// SIMATIC STEP 7 (V5.x) project Bai2_PLC

ORGANIZATION_BLOCK OB 1
TITLE = "Main Program Sweep (Cycle)"
VERSION : 0.1
VAR_TEMP
  OB1_EV_CLASS : BYTE ;	//Bits 0-3 = 1 (Coming event), Bits 4-7 = 1 (Event class 1)
  OB1_SCAN_1 : BYTE ;	//1 (Cold restart scan 1 of OB 1), 3 (Scan 2-n of OB 1)
  OB1_PRIORITY : BYTE ;	//Priority of OB Execution
  OB1_OB_NUMBR : BYTE ;	//1 (Organization block 1, OB1)
  OB1_RESERVED_1 : BYTE ;	//Reserved for system
  OB1_RESERVED_2 : BYTE ;	//Reserved for system
  OB1_PREV_CYCLE : INT ;	//Cycle time of previous OB1 scan (milliseconds)
  OB1_MIN_CYCLE : INT ;	//Minimum cycle time of OB1 (milliseconds)
  OB1_MAX_CYCLE : INT ;	//Maximum cycle time of OB1 (milliseconds)
  OB1_DATE_TIME : DATE_AND_TIME ;	//Date and time OB1 started
END_VAR
BEGIN
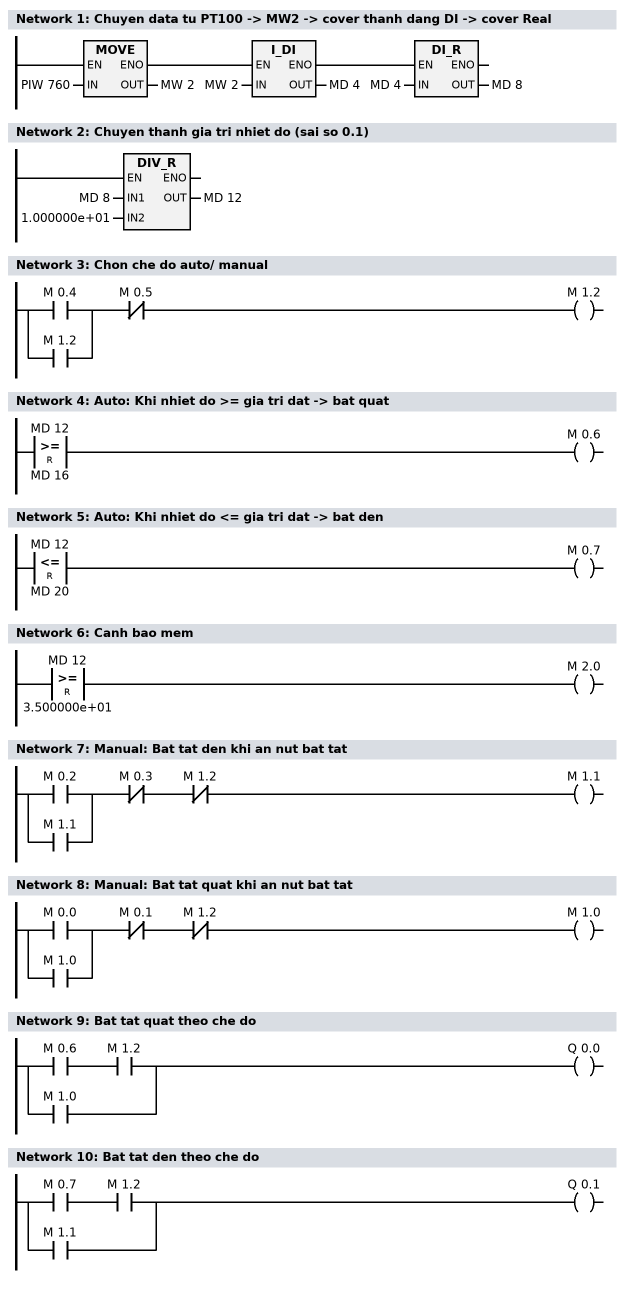
NETWORK
TITLE = Chuyen data tu PT100 -> MW2 -> cover thanh dang DI -> cover Real
      A(;
      A(;
      L     PIW 760;
      T     MW 2;
      SET;
      SAVE;
      CLR;
      A     BR;
      );
      JNB   _001;
      L     MW 2;
      ITD;
      T     MD 4;
      SET;
      SAVE;
      CLR;
_001: A     BR;
      );
      JNB   _002;
      L     MD 4;
      DTR;
      T     MD 8;
_002: NOP   0;
NETWORK
TITLE = Chuyen thanh gia tri nhiet do (sai so 0.1)
      L     MD 8;
      L     1.000000e+01;
      /R;
      T     MD 12;
      NOP   0;
NETWORK
TITLE = Chon che do auto/ manual
      A(;
      O     M 0.4;
      O     M 1.2;
      );
      AN    M 0.5;
      =     M 1.2;
NETWORK
TITLE = Auto: Khi nhiet do >= gia tri dat -> bat quat
      L     MD 12;
      L     MD 16;
      >=R;
      =     M 0.6;
NETWORK
TITLE = Auto: Khi nhiet do <= gia tri dat -> bat den
      L     MD 12;
      L     MD 20;
      <=R;
      =     M 0.7;
NETWORK
TITLE = Canh bao mem
      L     MD 12;
      L     3.500000e+01;
      >=R;
      =     M 2.0;
NETWORK
TITLE = Manual: Bat tat den khi an nut bat tat
      A(;
      O     M 0.2;
      O     M 1.1;
      );
      AN    M 0.3;
      AN    M 1.2;
      =     M 1.1;
NETWORK
TITLE = Manual: Bat tat quat khi an nut bat tat
      A(;
      O     M 0.0;
      O     M 1.0;
      );
      AN    M 0.1;
      AN    M 1.2;
      =     M 1.0;
NETWORK
TITLE = Bat tat quat theo che do
      A     M 0.6;
      A     M 1.2;
      O     M 1.0;
      =     Q 0.0;
NETWORK
TITLE = Bat tat den theo che do
      A     M 0.7;
      A     M 1.2;
      O     M 1.1;
      =     Q 0.1;
END_ORGANIZATION_BLOCK
